// TIA Portal V20 export
VAR_GLOBAL   // PLC tag table "Spare"
   "BA030AZSSP201.03" AT %I700.3 : Bool;   // SPARE
   "BA030AZSSP201.04" AT %I700.4 : Bool;   // SPARE
   "BA030AZSSP201.05" AT %I700.5 : Bool;   // SPARE
   "BA030AZSSP201.06" AT %I700.6 : Bool;   // SPARE
   "BA030AZSSP201.07" AT %I700.7 : Bool;   // SPARE
   "BA030AZSSP201.11" AT %I701.1 : Bool;   // SPARE
   "BA030AZSSP201.12" AT %I701.2 : Bool;   // SPARE
   "BA030AZSSP201.13" AT %I701.3 : Bool;   // SPARE
   "BA030AZSSP201.14" AT %I701.4 : Bool;   // SPARE
   "BA030AZSSP201.15" AT %I701.5 : Bool;   // SPARE
   "BA030AZSSP201.16" AT %I701.6 : Bool;   // SPARE
   "BA030AZSSP201.17" AT %I701.7 : Bool;   // SPARE
   "BA030AZSBK01.02" AT %I1000.2 : Bool;   // SPARE
   "BA030AZSBK01.06" AT %I1000.6 : Bool;   // SPARE
   "BA030AZSBK01.12" AT %I1001.2 : Bool;   // SPARE
   "BA030AZSBK01.14" AT %I1001.4 : Bool;   // SPARE
   "BA030AZSBK01.16" AT %I1001.6 : Bool;   // SPARE
   "BA030AZSBK01.17" AT %I1001.7 : Bool;   // SPARE
   "BA030AZSBK02.07" AT %I1004.7 : Bool;   // SPARE
   "BA030AZSBK02.17" AT %I1005.7 : Bool;   // SPARE
   "BA030AZSBK03.07" AT %I1008.7 : Bool;   // SPARE
   "BA030AZSBK04.11" AT %I1013.1 : Bool;   // SPARE
   "BA030AZSBK04.13" AT %I1013.3 : Bool;   // SPARE
   "BA030AZSBK04.15" AT %I1013.5 : Bool;   // SPARE
   "BA030AZSBK04.17" AT %I1013.7 : Bool;   // SPARE
   "BA030AZSBK05.11" AT %I1017.1 : Bool;   // SPARE
   "BA030AZSBK05.13" AT %I1017.3 : Bool;   // SPARE
   "BA030AZSBK05.15" AT %I1017.5 : Bool;   // SPARE
   "BA030AZSBK05.17" AT %I1017.7 : Bool;   // SPARE
   "BA030AZSBK06.05" AT %I1020.5 : Bool;   // SPARE
   "BA030AZSBK06.06" AT %I1020.6 : Bool;   // SPARE
   "BA030AZSBK06.07" AT %I1020.7 : Bool;   // SPARE
   "BA030AZSBK07.11" AT %I1025.1 : Bool;   // SPARE
   "BA030AZSBK07.13" AT %I1025.3 : Bool;   // SPARE
   "BA030AZSBK07.15" AT %I1025.5 : Bool;   // SPARE
   "BA030AZSBK07.17" AT %I1025.7 : Bool;   // SPARE
   "BA030AZSBK08.05" AT %I1028.5 : Bool;   // SPARE
   "BA030AZSBK08.06" AT %I1028.6 : Bool;   // SPARE
   "BA030AZSBK08.07" AT %I1028.7 : Bool;   // SPARE
   "BA030AZSBK09.11" AT %I1033.1 : Bool;   // SPARE
   "BA030AZSBK09.13" AT %I1033.3 : Bool;   // SPARE
   "BA030AZSBK09.15" AT %I1033.5 : Bool;   // SPARE
   "BA030AZSBK09.16" AT %I1033.6 : Bool;   // SPARE
   "BA030AZSBK09.17" AT %I1033.7 : Bool;   // SPARE
   "BA030AZSBK10.05" AT %I1036.5 : Bool;   // SPARE
   "BA030AZSBK10.06" AT %I1036.6 : Bool;   // SPARE
   "BA030AZSBK10.07" AT %I1036.7 : Bool;   // SPARE
   "BA030AZSBK10.13" AT %I1037.3 : Bool;   // SPARE
   "BA030AZSBK10.14" AT %I1037.4 : Bool;   // SPARE
   "BA030AZSBK10.15" AT %I1037.5 : Bool;   // SPARE
   "BA030AZSBK10.16" AT %I1037.6 : Bool;   // SPARE
   "BA030AZSBK10.17" AT %I1037.7 : Bool;   // SPARE
   "BA030AZSBK11.07" AT %I1040.7 : Bool;   // SPARE
   "BA030AZSBK12.01" AT %I1044.1 : Bool;   // SPARE
   "BA030AZSBK12.03" AT %I1044.3 : Bool;   // SPARE
   "BA030AZSBK12.05" AT %I1044.5 : Bool;   // SPARE
   "BA030AZSBK12.07" AT %I1044.7 : Bool;   // SPARE
   "BA030AZSBK12.11" AT %I1045.1 : Bool;   // SPARE
   "BA030AZSBK12.13" AT %I1045.3 : Bool;   // SPARE
   "BA030AZSBK12.15" AT %I1045.5 : Bool;   // SPARE
   "BA030AZSBK12.17" AT %I1045.7 : Bool;   // SPARE
   "BA030AZSBK13.11" AT %I1049.1 : Bool;   // SPARE
   "BA030AZSBK13.13" AT %I1049.3 : Bool;   // SPARE
   "BA030AZSBK13.15" AT %I1049.5 : Bool;   // SPARE
   "BA030AZSBK13.16" AT %I1049.6 : Bool;   // SPARE
   "BA030AZSBK13.17" AT %I1049.7 : Bool;   // SPARE
   "BA030AZSBK14.05" AT %I1052.5 : Bool;   // SPARE
   "BA030AZSBK14.06" AT %I1052.6 : Bool;   // SPARE
   "BA030AZSBK14.07" AT %I1052.7 : Bool;   // SPARE
   "BA030AZSBK14.13" AT %I1053.3 : Bool;   // SPARE
   "BA030AZSBK14.14" AT %I1053.4 : Bool;   // SPARE
   "BA030AZSBK14.15" AT %I1053.5 : Bool;   // SPARE
   "BA030AZSBK14.16" AT %I1053.6 : Bool;   // SPARE
   "BA030AZSBK14.17" AT %I1053.7 : Bool;   // SPARE
   "BA030AZSBK15.06" AT %I1056.6 : Bool;   // SPARE
   "BA030AZSBK15.07" AT %I1056.7 : Bool;   // RESERVE
   "BA030AZSBK16.01" AT %I1060.1 : Bool;   // SPARE
   "BA030AZSBK16.03" AT %I1060.3 : Bool;   // SPARE
   "BA030AZSBK16.05" AT %I1060.5 : Bool;   // SPARE
   "BA030AZSBK16.07" AT %I1060.7 : Bool;   // SPARE
   "BA030AZSBK16.11" AT %I1061.1 : Bool;   // SPARE
   "BA030AZSBK16.13" AT %I1061.3 : Bool;   // SPARE
   "BA030AZSBK16.15" AT %I1061.5 : Bool;   // SPARE
   "BA030AZSBK16.17" AT %I1061.7 : Bool;   // SPARE
   "BA030AZSBK17.03" AT %I1064.3 : Bool;   // SPARE
   "BA030AZSBK17.07" AT %I1064.7 : Bool;   // SPARE
   "BA030AZSBK18.11" AT %I1069.1 : Bool;   // SPARE
   "BA030AZSBK18.13" AT %I1069.3 : Bool;   // SPARE
   "BA030AZSBK18.15" AT %I1069.5 : Bool;   // SPARE
   "BA030AZSBK18.17" AT %I1069.7 : Bool;   // SPARE
   "BA030AZSBK19.11" AT %I1073.1 : Bool;   // SPARE
   "BA030AZSBK19.13" AT %I1073.3 : Bool;   // SPARE
   "BA030AZSBK19.15" AT %I1073.5 : Bool;   // SPARE
   "BA030AZSBK19.17" AT %I1073.7 : Bool;   // SPARE
   "BA030AZSBK20.11" AT %I1077.1 : Bool;   // SPARE
   "BA030AZSBK20.12" AT %I1077.2 : Bool;   // SPARE
   "BA030AZSBK20.13" AT %I1077.3 : Bool;   // SPARE
   "BA030AZSBK21.03" AT %I1080.3 : Bool;   // SPARE
   "BA030AZSBK21.07" AT %I1080.7 : Bool;   // SPARE
   "BA030AZSBK22.01" AT %I1084.1 : Bool;   // SPARE
   "BA030AZSBK22.11" AT %I1085.1 : Bool;   // SPARE
   "BA030AZSBK22.12" AT %I1085.2 : Bool;   // SPARE
   "BA030AZSBK22.17" AT %I1085.7 : Bool;   // SPARE
   "BA030AZSBK23.03" AT %I1088.3 : Bool;   // SPARE
   "BA030AZSBK23.04" AT %I1088.4 : Bool;   // SPARE
   "BA030AZSBK23.05" AT %I1088.5 : Bool;   // SPARE
   "BA030AZSBK23.07" AT %I1088.7 : Bool;   // SPARE
   "BA030AZSBK23.11" AT %I1089.1 : Bool;   // SPARE
   "BA030AZSBK23.13" AT %I1089.3 : Bool;   // SPARE
   "BA030AZSBK23.14" AT %I1089.4 : Bool;   // SPARE
   "BA030AZSBK23.15" AT %I1089.5 : Bool;   // SPARE
   "BA030AZSBK23.16" AT %I1089.6 : Bool;   // SPARE
   "BA030AZSBK23.17" AT %I1089.7 : Bool;   // SPARE
   "BA030AZSBK24.01" AT %I1092.1 : Bool;   // SPARE
   "BA030AZSBK24.03" AT %I1092.3 : Bool;   // SPARE
   "BA030AZSBK24.05" AT %I1092.5 : Bool;   // SPARE
   "BA030AZSBK24.07" AT %I1092.7 : Bool;   // SPARE
   "BA030AZSBK24.11" AT %I1093.1 : Bool;   // SPARE
   "BA030AZSBK24.13" AT %I1093.3 : Bool;   // SPARE
   "BA030AZSBK24.15" AT %I1093.5 : Bool;   // SPARE
   "BA030AZSBK24.17" AT %I1093.7 : Bool;   // SPARE
   "BA030AZSBK25.07" AT %I1096.7 : Bool;   // SPARE
   "BA030AZSBK26.04" AT %I1100.4 : Bool;   // SPARE
   "BA030AZSBK26.06" AT %I1100.6 : Bool;   // SPARE
   "BA030AZSBK26.07" AT %I1100.7 : Bool;   // SPARE
   "BA030AZSBK26.10" AT %I1101.0 : Bool;   // SPARE
   "BA030AZSBK26.14" AT %I1101.4 : Bool;   // SPARE
   "BA030AZSBK26.16" AT %I1101.6 : Bool;   // SPARE
   "BA030AZSBK26.17" AT %I1101.7 : Bool;   // SPARE
   "BA030AZSBK27.00" AT %I1104.0 : Bool;   // SPARE
   "BA030AZSBK27.02" AT %I1104.2 : Bool;   // SPARE
   "BA030AZSBK27.04" AT %I1104.4 : Bool;   // SPARE
   "BA030AZSBK27.07" AT %I1104.7 : Bool;   // SPARE
   "BA030AZSBK27.10" AT %I1105.0 : Bool;   // SPARE
   "BA030AZSBK27.12" AT %I1105.2 : Bool;   // SPARE
   "BA030AZSBK27.14" AT %I1105.4 : Bool;   // SPARE
   "BA030AZSBK27.16" AT %I1105.6 : Bool;   // SPARE
   "BA030AZSBK27.17" AT %I1105.7 : Bool;   // SPARE
   "BA030AZSBK28.04" AT %I1108.4 : Bool;   // SPARE
   "BA030AZSBK28.05" AT %I1108.5 : Bool;   // SPARE
   "BA030AZSBK28.07" AT %I1108.7 : Bool;   // SPARE
   "BA030AZSSP501.12" AT %I3001.2 : Bool;   // SPARE
   "BA030AZSSP501.13" AT %I3001.3 : Bool;   // SPARE
   "BA030AZSSP501.16" AT %I3001.6 : Bool;   // SPARE
   "BA030AZSSP501.17" AT %I3001.7 : Bool;   // SPARE
   "BA030AZSPM01.03" AT %Q2000.3 : Bool;   // SPARE
   "BA030AZSPM01.05" AT %Q2000.5 : Bool;   // SPARE
   "BA030AZSPM01.20" AT %Q2002.0 : Bool;   // SPARE
   "BA030AZSPM01.21" AT %Q2002.1 : Bool;   // SPARE
   "BA030AZSPM01.22" AT %Q2002.2 : Bool;   // SPARE
   "BA030AZSPM01.23" AT %Q2002.3 : Bool;   // SPARE
   "BA030AZSPM01.24" AT %Q2002.4 : Bool;   // SPARE
   "BA030AZSPM01.25" AT %Q2002.5 : Bool;   // SPARE
   "BA030AZSPM01.26" AT %Q2002.6 : Bool;   // SPARE
   "BA030AZSPM01.27" AT %Q2002.7 : Bool;   // SPARE
   "BA030AZSPM01.30" AT %Q2003.0 : Bool;   // SPARE
   "BA030AZSPM01.31" AT %Q2003.1 : Bool;   // SPARE
   "BA030AZSPM01.32" AT %Q2003.2 : Bool;   // SPARE
   "BA030AZSPM01.33" AT %Q2003.3 : Bool;   // SPARE
   "BA030AZSPM01.34" AT %Q2003.4 : Bool;   // SPARE
   "BA030AZSPM01.35" AT %Q2003.5 : Bool;   // SPARE
   "BA030AZSPM01.36" AT %Q2003.6 : Bool;   // SPARE
   "BA030AZSPM01.37" AT %Q2003.7 : Bool;   // SPARE
   "BA030AZSPM02.16" AT %Q2005.6 : Bool;   // SPARE
   "BA030AZSPM02.17" AT %Q2005.7 : Bool;   // SPARE
   "BA030AZSPM02.20" AT %Q2006.0 : Bool;   // SPARE
   "BA030AZSPM02.21" AT %Q2006.1 : Bool;   // SPARE
   "BA030AZSPM02.22" AT %Q2006.2 : Bool;   // SPARE
   "BA030AZSPM02.23" AT %Q2006.3 : Bool;   // SPARE
   "BA030AZSPM02.24" AT %Q2006.4 : Bool;   // SPARE
   "BA030AZSPM02.25" AT %Q2006.5 : Bool;   // SPARE
   "BA030AZSPM02.26" AT %Q2006.6 : Bool;   // SPARE
   "BA030AZSPM02.27" AT %Q2006.7 : Bool;   // SPARE
   "BA030AZSPM02.30" AT %Q2007.0 : Bool;   // SPARE
   "BA030AZSPM02.31" AT %Q2007.1 : Bool;   // SPARE
   "BA030AZSPM02.32" AT %Q2007.2 : Bool;   // SPARE
   "BA030AZSPM02.33" AT %Q2007.3 : Bool;   // SPARE
   "BA030AZSPM02.34" AT %Q2007.4 : Bool;   // SPARE
   "BA030AZSPM02.35" AT %Q2007.5 : Bool;   // SPARE
   "BA030AZSPM02.36" AT %Q2007.6 : Bool;   // SPARE
   "BA030AZSPM02.37" AT %Q2007.7 : Bool;   // SPARE
   "BA030AZSPM03.16" AT %Q2009.6 : Bool;   // SPARE
   "BA030AZSPM03.17" AT %Q2009.7 : Bool;   // SPARE
   "BA030AZSPM03.20" AT %Q2010.0 : Bool;   // SPARE
   "BA030AZSPM03.21" AT %Q2010.1 : Bool;   // SPARE
   "BA030AZSPM03.22" AT %Q2010.2 : Bool;   // SPARE
   "BA030AZSPM03.23" AT %Q2010.3 : Bool;   // SPARE
   "BA030AZSPM03.24" AT %Q2010.4 : Bool;   // SPARE
   "BA030AZSPM03.25" AT %Q2010.5 : Bool;   // SPARE
   "BA030AZSPM03.26" AT %Q2010.6 : Bool;   // SPARE
   "BA030AZSPM03.27" AT %Q2010.7 : Bool;   // SPARE
   "BA030AZSPM03.30" AT %Q2011.0 : Bool;   // SPARE
   "BA030AZSPM03.31" AT %Q2011.1 : Bool;   // SPARE
   "BA030AZSPM03.32" AT %Q2011.2 : Bool;   // SPARE
   "BA030AZSPM03.33" AT %Q2011.3 : Bool;   // SPARE
   "BA030AZSPM03.34" AT %Q2011.4 : Bool;   // SPARE
   "BA030AZSPM03.35" AT %Q2011.5 : Bool;   // SPARE
   "BA030AZSPM03.36" AT %Q2011.6 : Bool;   // SPARE
   "BA030AZSPM03.37" AT %Q2011.7 : Bool;   // SPARE
   "BA030AZSPM04.03" AT %Q2012.3 : Bool;   // SPARE
   "BA030AZSPM04.05" AT %Q2012.5 : Bool;   // SPARE
   "BA030AZSPM04.07" AT %Q2012.7 : Bool;   // SPARE
   "BA030AZSPM04.11" AT %Q2013.1 : Bool;   // SPARE
   "BA030AZSPM04.12" AT %Q2013.2 : Bool;   // SPARE
   "BA030AZSPM04.13" AT %Q2013.3 : Bool;   // SPARE
   "BA030AZSPM04.14" AT %Q2013.4 : Bool;   // SPARE
   "BA030AZSPM04.15" AT %Q2013.5 : Bool;   // SPARE
   "BA030AZSPM04.16" AT %Q2013.6 : Bool;   // SPARE
   "BA030AZSPM04.17" AT %Q2013.7 : Bool;   // SPARE
   "BA030AZSPM04.20" AT %Q2014.0 : Bool;   // SPARE
   "BA030AZSPM04.21" AT %Q2014.1 : Bool;   // SPARE
   "BA030AZSPM04.22" AT %Q2014.2 : Bool;   // SPARE
   "BA030AZSPM04.23" AT %Q2014.3 : Bool;   // SPARE
   "BA030AZSPM04.24" AT %Q2014.4 : Bool;   // SPARE
   "BA030AZSPM04.25" AT %Q2014.5 : Bool;   // SPARE
   "BA030AZSPM04.26" AT %Q2014.6 : Bool;   // SPARE
   "BA030AZSPM04.27" AT %Q2014.7 : Bool;   // SPARE
   "BA030AZSPM04.30" AT %Q2015.0 : Bool;   // SPARE
   "BA030AZSPM04.31" AT %Q2015.1 : Bool;   // SPARE
   "BA030AZSPM04.32" AT %Q2015.2 : Bool;   // SPARE
   "BA030AZSPM04.33" AT %Q2015.3 : Bool;   // SPARE
   "BA030AZSPM04.34" AT %Q2015.4 : Bool;   // SPARE
   "BA030AZSPM04.35" AT %Q2015.5 : Bool;   // SPARE
   "BA030AZSPM04.36" AT %Q2015.6 : Bool;   // SPARE
   "BA030AZSPM04.37" AT %Q2015.7 : Bool;   // SPARE
   "BA030AZSPM05.01" AT %Q2016.1 : Bool;   // SPARE
   "BA030AZSPM05.20" AT %Q2018.0 : Bool;   // SPARE
   "BA030AZSPM05.21" AT %Q2018.1 : Bool;   // SPARE
   "BA030AZSPM05.22" AT %Q2018.2 : Bool;   // SPARE
   "BA030AZSPM05.23" AT %Q2018.3 : Bool;   // SPARE
   "BA030AZSPM05.24" AT %Q2018.4 : Bool;   // SPARE
   "BA030AZSPM05.25" AT %Q2018.5 : Bool;   // SPARE
   "BA030AZSPM05.26" AT %Q2018.6 : Bool;   // SPARE
   "BA030AZSPM05.27" AT %Q2018.7 : Bool;   // SPARE
   "BA030AZSPM05.30" AT %Q2019.0 : Bool;   // SPARE
   "BA030AZSPM05.31" AT %Q2019.1 : Bool;   // SPARE
   "BA030AZSPM05.32" AT %Q2019.2 : Bool;   // SPARE
   "BA030AZSPM05.33" AT %Q2019.3 : Bool;   // SPARE
   "BA030AZSPM05.34" AT %Q2019.4 : Bool;   // SPARE
   "BA030AZSPM05.35" AT %Q2019.5 : Bool;   // SPARE
   "BA030AZSPM05.36" AT %Q2019.6 : Bool;   // SPARE
   "BA030AZSPM05.37" AT %Q2019.7 : Bool;   // SPARE
   "BA030AZSPM06.01" AT %Q2020.1 : Bool;   // SPARE
   "BA030AZSPM06.22" AT %Q2022.2 : Bool;   // SPARE
   "BA030AZSPM06.23" AT %Q2022.3 : Bool;   // SPARE
   "BA030AZSPM06.24" AT %Q2022.4 : Bool;   // SPARE
   "BA030AZSPM06.25" AT %Q2022.5 : Bool;   // SPARE
   "BA030AZSPM06.26" AT %Q2022.6 : Bool;   // SPARE
   "BA030AZSPM06.27" AT %Q2022.7 : Bool;   // SPARE
   "BA030AZSPM06.30" AT %Q2023.0 : Bool;   // SPARE
   "BA030AZSPM06.31" AT %Q2023.1 : Bool;   // SPARE
   "BA030AZSPM06.32" AT %Q2023.2 : Bool;   // SPARE
   "BA030AZSPM06.33" AT %Q2023.3 : Bool;   // SPARE
   "BA030AZSPM06.34" AT %Q2023.4 : Bool;   // SPARE
   "BA030AZSPM06.35" AT %Q2023.5 : Bool;   // SPARE
   "BA030AZSPM06.36" AT %Q2023.6 : Bool;   // SPARE
   "BA030AZSPM06.37" AT %Q2023.7 : Bool;   // SPARE
   "BA030AZSPM07.22" AT %Q2026.2 : Bool;   // SPARE
   "BA030AZSPM07.23" AT %Q2026.3 : Bool;   // SPARE
   "BA030AZSPM07.24" AT %Q2026.4 : Bool;   // SPARE
   "BA030AZSPM07.25" AT %Q2026.5 : Bool;   // SPARE
   "BA030AZSPM07.26" AT %Q2026.6 : Bool;   // SPARE
   "BA030AZSPM07.27" AT %Q2026.7 : Bool;   // SPARE
   "BA030AZSPM07.30" AT %Q2027.0 : Bool;   // SPARE
   "BA030AZSPM07.31" AT %Q2027.1 : Bool;   // SPARE
   "BA030AZSPM07.32" AT %Q2027.2 : Bool;   // SPARE
   "BA030AZSPM07.33" AT %Q2027.3 : Bool;   // SPARE
   "BA030AZSPM07.34" AT %Q2027.4 : Bool;   // SPARE
   "BA030AZSPM07.35" AT %Q2027.5 : Bool;   // SPARE
   "BA030AZSPM07.36" AT %Q2027.6 : Bool;   // SPARE
   "BA030AZSPM07.37" AT %Q2027.7 : Bool;   // SPARE
   "BA030AZSBK30.06" AT %Q2104.6 : Bool;   // SPARE
   "BA030AZSBK30.07" AT %Q2104.7 : Bool;   // SPARE
   "BA030AZSSP202.05" AT %Q700.5 : Bool;   // SPARE
   "BA030AZSSP202.06" AT %Q700.6 : Bool;   // SPARE
   "BA030AZSSP202.07" AT %Q700.7 : Bool;   // SPARE
   "BA030AZSSP502.01" AT %Q3000.1 : Bool;   // SPARE
   "BA030AZSSP502.02" AT %Q3000.2 : Bool;   // SPARE
   "BA030AZSSP502.03" AT %Q3000.3 : Bool;   // SPARE
   "BA030AZSSP502.04" AT %Q3000.4 : Bool;   // SPARE
   "BA030AZSSP502.05" AT %Q3000.5 : Bool;   // SPARE
   "BA030AZSSP502.06" AT %Q3000.6 : Bool;   // SPARE
   "BA030AZSSP502.07" AT %Q3000.7 : Bool;   // SPARE
   "BA030AZSSP502.12" AT %Q3001.2 : Bool;   // SPARE
   "BA030AZSSP502.13" AT %Q3001.3 : Bool;   // SPARE
   "BA030AZSSP502.16" AT %Q3001.6 : Bool;   // SPARE
   "BA030AZSSP502.17" AT %Q3001.7 : Bool;   // SPARE
   "BA030AZSBK20.17" AT %I1077.7 : Bool;   // SPARE
   "BA030AZSBK20.07" AT %I1076.7 : Bool;   // SPARE
   "BA030AZSBK34.02" AT %IW2216 : Int;   // SPARE
   "BA030AZSBK34.03" AT %IW2218 : Int;   // SPARE
   "BA030AZSBK34.04" AT %IW2220 : Int;   // SPARE
   "BA030AZSBK34.05" AT %IW2222 : Int;   // SPARE
   "BA030AZSMP101.00" AT %I100.0 : Bool;   // SPARE
   "BA030AZSMP101.01" AT %I100.1 : Bool;   // SPARE
   "BA030AZSMP101.05" AT %I100.5 : Bool;   // SPARE
   "BA030AZSMP101.10" AT %I101.0 : Bool;   // SPARE
   "BA030AZSMP101.12" AT %I101.2 : Bool;   // SPARE
   "BA030AZSMP101.21" AT %I102.1 : Bool;   // SPARE
   "BA030AZSMP101.22" AT %I102.2 : Bool;   // SPARE
   "BA030AZSMP101.30" AT %I103.0 : Bool;   // SPARE
   "BA030AZSMP101.32" AT %I103.2 : Bool;   // SPARE
   "BA030AZSMP102.05" AT %I104.5 : Bool;   // SPARE
   "BA030AZSMP102.10" AT %I105.0 : Bool;   // SPARE
   "BA030AZSMP102.23" AT %I106.3 : Bool;   // SPARE
   "BA030AZSBK01.05" AT %I1000.5 : Bool;   // SPARE
   "BA030AZSBK01.15" AT %I1001.5 : Bool;   // SPARE
   "BA030AZSBK05.04" AT %I1016.4 : Bool;   // SPARE
   "BA030AZSBK05.14" AT %I1017.4 : Bool;   // SPARE
   "BA030AZSBK07.04" AT %I1024.4 : Bool;   // SPARE
   "BA030AZSBK07.14" AT %I1025.4 : Bool;   // SPARE
   "BA030AZSBK11.01" AT %I1040.1 : Bool;   // RESERVE
   "BA030AZSBK20.15" AT %I1077.5 : Bool;   // SPARE
   "BA030AZSBK22.15" AT %I1085.5 : Bool;   // SPARE
   "BA030AZSBK25.03" AT %I1096.3 : Bool;   // SPARE
   "BA030AZSSP508.06" AT %I3002.6 : Bool;   // SPARE
   "BA030AZSSP508.07" AT %I3002.7 : Bool;   // SPARE
   "BA030AZSSP508.10" AT %I3003.0 : Bool;   // SPARE
   "BA030AZSSP508.11" AT %I3003.1 : Bool;   // SPARE
   "BA030AZSSP508.12" AT %I3003.2 : Bool;   // SPARE
   "BA030AZSSP508.13" AT %I3003.3 : Bool;   // SPARE
   "BA030AZSSP508.14" AT %I3003.4 : Bool;   // SPARE
   "BA030AZSSP508.15" AT %I3003.5 : Bool;   // SPARE
   "BA030AZSSP508.16" AT %I3003.6 : Bool;   // SPARE
   "BA030AZSSP508.17" AT %I3003.7 : Bool;   // SPARE
   "BA030AZSSP503.01" AT %IW3102 : Int;   // SPARE
   "BA030AZSSP503.02" AT %IW3104 : Int;   // SPARE
   "BA030AZSSP503.03" AT %IW3106 : Int;   // SPARE
   "BA030AZSSP513.01" AT %IW3110 : Int;   // SPARE
   "BA030AZSSP504.00" AT %I3300.0 : Bool;   // SPARE
   "BA030AZSSP504.01" AT %I3300.1 : Bool;   // SPARE
   "BA030AZSSP504.02" AT %I3300.2 : Bool;   // SPARE
   "BA030AZSSP504.03" AT %I3300.3 : Bool;   // SPARE
   "BA030AZSSP505.00" AT %I3350.0 : Bool;   // SPARE
   "BA030AZSSP505.01" AT %I3350.1 : Bool;   // SPARE
   "BA030AZSSP505.02" AT %I3350.2 : Bool;   // SPARE
   "BA030AZSSP505.03" AT %I3350.3 : Bool;   // SPARE
   "BA030AZSMP104.00" AT %Q100.0 : Bool;   // SPARE
   "BA030AZSMP104.01" AT %Q100.1 : Bool;   // SPARE
   "BA030AZSMP104.02" AT %Q100.2 : Bool;   // SPARE
   "BA030AZSMP104.04" AT %Q100.4 : Bool;   // SPARE
   "BA030AZSMP104.05" AT %Q100.5 : Bool;   // SPARE
   "BA030AZSMP104.06" AT %Q100.6 : Bool;   // SPARE
   "BA030AZSMP104.07" AT %Q100.7 : Bool;   // SPARE
   "BA030AZSSP202.16" AT %Q701.6 : Bool;   // SPARE
   "BA030AZSPM01.12" AT %Q2001.2 : Bool;   // SPARE
   "BA030AZSPM01.13" AT %Q2001.3 : Bool;   // SPARE
   "BA030AZSPM01.15" AT %Q2001.5 : Bool;   // SPARE
   "BA030AZSPM01.17" AT %Q2001.7 : Bool;   // SPARE
   "BA030AZSPM07.10" AT %Q2025.0 : Bool;   // SPARE
   "BA030AZSPM07.11" AT %Q2025.1 : Bool;   // SPARE
   "BA030AZSBK33.00" AT %Q2208.0 : Bool;   // SPARE
   "BA030AZSBK33.01" AT %Q2208.1 : Bool;   // SPARE
   "BA030AZSBK33.02" AT %Q2208.2 : Bool;   // SPARE
   "BA030AZSBK33.03" AT %Q2208.3 : Bool;   // SPARE
   "BA030AZSBK33.04" AT %Q2208.4 : Bool;   // SPARE
   "BA030AZSBK33.05" AT %Q2208.5 : Bool;   // SPARE
   "BA030AZSBK33.06" AT %Q2208.6 : Bool;   // SPARE
   "BA030AZSBK33.07" AT %Q2208.7 : Bool;   // SPARE
   "BA030AZSBK34.11" AT %QW2214 : Int;   // SPARE
   "BA030AZSSP504.10" AT %Q3300.0 : Bool;   // SPARE
   "BA030AZSSP504.11" AT %Q3300.1 : Bool;   // SPARE
   "BA030AZSSP504.15" AT %Q3300.5 : Bool;   // SPARE
   "BA030AZSSP505.10" AT %Q3350.0 : Bool;   // SPARE
   "BA030AZSSP505.11" AT %Q3350.1 : Bool;   // SPARE
   "BA030AZSSP505.12" AT %Q3350.2 : Bool;   // SPARE
   "BA030AZSSP505.13" AT %Q3350.3 : Bool;   // SPARE
   "BA030AZSSP505.14" AT %Q3350.4 : Bool;   // SPARE
   "BA030AZSSP505.15" AT %Q3350.5 : Bool;   // SPARE
   "BA030AZSMP103.30" AT %I111.0 : Bool;   // SPARE
   "BA030AZSMP103.27" AT %I110.7 : Bool;   // SPARE
   "BA030AZSMP103.26" AT %I110.6 : Bool;   // SPARE
   "BA030AZSMP103.25" AT %I110.5 : Bool;   // SPARE
   "BA030AZSMP103.24" AT %I110.4 : Bool;   // SPARE
   "BA030AZSMP103.23" AT %I110.3 : Bool;   // SPARE
   "BA030AZSMP103.22" AT %I110.2 : Bool;   // SPARE
   "BA030AZSMP103.10" AT %I109.0 : Bool;   // SPARE
   "BA030AZSMP103.17" AT %I109.7 : Bool;   // SPARE
   "BA030AZSMP103.21" AT %I110.1 : Bool;   // SPARE
   "BA030AZSMP103.16" AT %I109.6 : Bool;   // SPARE
   "BA030AZSMP103.20" AT %I110.0 : Bool;   // SPARE
   "BA030AZSMP103.11" AT %I109.1 : Bool;   // SPARE
   "BA030AZSMP103.12" AT %I109.2 : Bool;   // SPARE
   "BA030AZSMP103.13" AT %I109.3 : Bool;   // SPARE
   "BA030AZSMP103.14" AT %I109.4 : Bool;   // SPARE
   "BA030AZSMP103.15" AT %I109.5 : Bool;   // SPARE
   "BA030AZSSP202.02" AT %Q700.2 : Bool;   // SPARE
   "BA030AZSMP103.07" AT %I108.7 : Bool;   // SPARE
   "BA030AZSMP104.10" AT %Q101.0 : Bool;   // SPARE
   "BA030AZSSP201.02" AT %I700.2 : Bool;   // RESERVE
   "BA030AZSSP202.17" AT %Q701.7 : Bool;   // SPARE
   "BA030AZSMP103.02" AT %I108.2 : Bool;   // SPARE
   "BA030AZSMP104.15" AT %Q101.5 : Bool;   // SPARE
   "BA030AZSMP104.16" AT %Q101.6 : Bool;   // SPARE
   "BA030AZSMP104.17" AT %Q101.7 : Bool;   // SPARE
   "BA030AZSMP104.20" AT %Q102.0 : Bool;   // SPARE
   "BA030AZSMP103.03" AT %I108.3 : Bool;   // SPARE
   "BA030AZSMP104.37" AT %Q103.7 : Bool;   // SPARE
   "BA030AZSMP104.34" AT %Q103.4 : Bool;   // SPARE
   "BA030AZSMP104.36" AT %Q103.6 : Bool;   // SPARE
   "BA030AZSMP104.35" AT %Q103.5 : Bool;   // SPARE
   "BA030AZSMP103.05" AT %I108.5 : Bool;   // SPARE
   "BA030AZSMP104.32" AT %Q103.2 : Bool;   // SPARE
   "BA030AZSMP104.33" AT %Q103.3 : Bool;   // SPARE
   "BA030AZSMP104.31" AT %Q103.1 : Bool;   // SPARE
   "BA030AZSMP104.30" AT %Q103.0 : Bool;   // SPARE
   "BA030AZSMP104.27" AT %Q102.7 : Bool;   // SPARE
   "BA030AZSMP104.26" AT %Q102.6 : Bool;   // SPARE
   "BA030AZSMP104.25" AT %Q102.5 : Bool;   // SPARE
   "BA030AZSMP104.24" AT %Q102.4 : Bool;   // SPARE
   "BA030AZSMP104.23" AT %Q102.3 : Bool;   // SPARE
   "BA030AZSMP104.22" AT %Q102.2 : Bool;   // SPARE
   "BA030AZSMP104.21" AT %Q102.1 : Bool;   // SPARE
   "BA030AZSMP103.37" AT %I111.7 : Bool;   // SPARE
   "BA030AZSMP103.36" AT %I111.6 : Bool;   // SPARE
   "BA030AZSMP103.35" AT %I111.5 : Bool;   // SPARE
   "BA030AZSMP103.31" AT %I111.1 : Bool;   // SPARE
   "BA030AZSMP103.34" AT %I111.4 : Bool;   // SPARE
   "BA030AZSMP103.33" AT %I111.3 : Bool;   // SPARE
   "BA030AZSMP103.32" AT %I111.2 : Bool;   // SPARE
   "BA030AZSBK34.06" AT %IW2224 : Word;   // SPARE
   "BA030AZSBK34.07" AT %IW2226 : Word;   // SPARE
END_VAR
